// TIA Portal V19 export
TYPE "CTRL_MTR"
   STRUCT
      status : Bool;
      sim : "UDT_SIM_MTR";
   END_STRUCT;
END_TYPE
